PROGRAM FnR_Switch
VAR
	qFNR : BOOL; //0 = user control, 1 = PLC controlled FNR
	qFNRDir : BOOL; //Sets direction 0 = reverse, 1 = forward
END_VAR

//Program to select what direction the car should go

IF MAIN.sCommand = 'Forward' THEN
	qFNR := TRUE;
	qFNRDir := TRUE;
ELSIF MAIN.sCommand = 'Reverse' THEN
	qFNR := TRUE;
	qFNRDir := FALSE;
ELSIF Main.sCommand = 'Manual' THEN //supposed to be manual mode
	qFNR := FALSE;
	qFNRDir := FALSE; //This one doesn't really matter
END_IF

END_PROGRAM

(* stored: Version 1.1.0.1, ProductVersion 3.1.4024.3
   POU FnR_Switch: Id {c8d29c2d-20b9-434a-9a27-d6db48306212}, SpecialFunc None *)
